FUNCTION_BLOCK FB_MotionInterlocksLimSw_TestDouble IMPLEMENTS I_MotionInterlocks
VAR
END_VAR

METHOD AxisStatus
VAR_INPUT
    HomeBusy	: BOOL;
    PositiveDirection	: BOOL;
    NegativeDirection	: BOOL;
END_VAR
END_METHOD

METHOD DriveCommands
VAR_INPUT
    MoveEnable: BOOL;
    NewMoveReq : BOOL;
END_VAR
END_METHOD

PROPERTY Error : BOOL
GET
END_GET
END_PROPERTY

PROPERTY ErrorID : UDINT
GET
END_GET
END_PROPERTY

{warning 'Add property implementation'}
PROPERTY HomeSensor : BOOL
GET
END_GET
END_PROPERTY

PROPERTY InterlockEvent : BOOL
GET
END_GET
END_PROPERTY

PROPERTY LimHome : BOOL
GET
END_GET
END_PROPERTY

PROPERTY Message : T_MAXSTRING
GET
END_GET
END_PROPERTY

PROPERTY MoveBackwardEnabled : BOOL
GET
END_GET
END_PROPERTY

PROPERTY MoveForwardEnabled : BOOL
GET
END_GET
END_PROPERTY

PROPERTY MoveOk : BOOL
GET
END_GET
END_PROPERTY

PROPERTY PowerEnabled : BOOL
GET
END_GET
END_PROPERTY

METHOD Reset
END_METHOD

PROPERTY Warning : BOOL
GET
END_GET
END_PROPERTY

END_FUNCTION_BLOCK

(* stored: Version 1.1.0.1
   POU FB_MotionInterlocksLimSw_TestDouble: Id {21f43876-bbfe-45b3-9c17-f49316824f4b}, SpecialFunc None
   Method AxisStatus: Id {50c5bd0b-cc66-4749-8282-e5e3388dc90e}
   Method DriveCommands: Id {33f79738-8853-40d3-b276-fd3ec975ee74}
   Property Error: Id {2d82a3f7-e9d9-4f60-89ee-f767c119473b}
   Get Get: Id {0c9adc32-875f-455a-9348-9e91c2136a2e}
   Property ErrorID: Id {7591664c-59d6-4ea6-ad7a-b681f08c6bcb}
   Get Get: Id {09b56839-3ecc-4575-9657-b30965a00f60}
   Property HomeSensor: Id {2760f0fe-2a1a-4add-9034-99f78bf03db8}
   Get Get: Id {1a71bd82-c6e8-4066-8710-c1c0e8e29cec}
   Property InterlockEvent: Id {462e9ab6-e8ad-4dc9-b9b7-9bd40388e72b}
   Get Get: Id {c25ec5f6-f6f9-4e64-8f34-2543ccad456d}
   Property LimHome: Id {996b3d94-6585-4089-bf52-671882c7dacd}
   Get Get: Id {6cf28804-ad65-4297-bb72-3dbdad554599}
   Property Message: Id {b505fe82-ef78-4450-b778-d2c5899646d2}
   Get Get: Id {dccbdb6b-766a-405b-95e8-5df32119c93f}
   Property MoveBackwardEnabled: Id {ed482ad7-b1c3-412c-b832-6da8fe190d69}
   Get Get: Id {67810e1e-6b2d-43ef-b25c-e51d48dcc777}
   Property MoveForwardEnabled: Id {3dea3059-8830-4c14-9c0d-196aba715801}
   Get Get: Id {7d4bfd5f-8649-4742-8367-f47786025327}
   Property MoveOk: Id {65cb5539-77ba-45bb-a7c8-e0a3eaedca97}
   Get Get: Id {55e9535f-457b-4dcc-9e51-a423b28cefb8}
   Property PowerEnabled: Id {d3350f4f-282b-492a-8e6d-573e2b2cca20}
   Get Get: Id {36d3dc3c-431d-4213-b2b1-505c852c4fc6}
   Method Reset: Id {d7213581-eb45-4db7-87f8-6dbc2af5c9c3}
   Property Warning: Id {08266c97-a963-44e9-976e-acb204a37e59}
   Get Get: Id {87c853ab-7d2a-4039-a7e5-d576f8c47535} *)
